INTERFACE I_ConveyerSection EXTENDS __SYSTEM.IQueryInterface

PROPERTY DwnStrmHndShkIn : BOOL
SET
END_SET
END_PROPERTY

PROPERTY DwnStrmHndShkOut : BOOL
GET
END_GET
END_PROPERTY

PROPERTY HMI : ARRAY[0..15] OF BOOL
GET
END_GET
END_PROPERTY

PROPERTY Id : UINT
GET
END_GET
SET
END_SET
END_PROPERTY

PROPERTY Pos : INT
GET
END_GET
SET
END_SET
END_PROPERTY

METHOD  Sequence : BOOL
VAR_INPUT
END_VAR
END_METHOD

METHOD startSequence : BOOL
VAR_INPUT
END_VAR
END_METHOD

METHOD stopSequence : BOOL
VAR_INPUT
END_VAR
END_METHOD

PROPERTY UpStrmHndShkIn : BOOL
SET
END_SET
END_PROPERTY

PROPERTY UpStrmHndShkOut : BOOL
GET
END_GET
END_PROPERTY

END_INTERFACE

(* stored: Version 1.1.0.1, ProductVersion 3.1.4024.6
   Itf I_ConveyerSection: Id {04d35945-385d-4123-9f2d-0739f05d8d7a}
   Property DwnStrmHndShkIn: Id {c188acd7-255a-464a-9ec1-1a7a647d59fe}
   Set Set: Id {1f5f4b12-5a3d-49e4-b953-36bb472f7c39}
   Property DwnStrmHndShkOut: Id {0c288d01-69ae-40ab-bd04-cec4de488d06}
   Get Get: Id {3dd57110-d022-4d7f-9835-f056523666b1}
   Property HMI: Id {14b95b79-30a2-4403-958e-3a413ec685e4}
   Get Get: Id {86ead9e8-1bb6-4423-9fad-524d3fadc868}
   Property Id: Id {d1169deb-72c7-4805-ad05-40dc16710016}
   Get Get: Id {a3d5a66a-749c-4c19-b6d0-65d283ddc20d}
   Set Set: Id {b121f4d3-40a8-4233-8949-e50f88a25dbc}
   Property Pos: Id {163d15c6-d9fe-441e-a293-f71f6cfda351}
   Get Get: Id {e165856c-5cfa-4fa1-b5b4-ea555dc55d47}
   Set Set: Id {d205e006-5608-4033-a16d-8b316a867f9c}
   Method Sequence: Id {afede655-2abb-4409-8510-a47763fd7f4c}
   Method startSequence: Id {4056de14-a7e2-450a-b73c-a88c86b2def7}
   Method stopSequence: Id {5b80c52f-6efe-4fee-89ab-84ec1a9d4f20}
   Property UpStrmHndShkIn: Id {dbd0dc8a-bfa3-43a9-bb38-0d9db277c5c5}
   Set Set: Id {a419933d-a7e4-4761-912e-7f9846f6bae7}
   Property UpStrmHndShkOut: Id {b5eceecb-2001-417e-9f79-881fadc4567d}
   Get Get: Id {5457ecda-8b58-4b67-9db7-1819519620a8} *)
